PROGRAM MAIN
VAR
	master,slave:					axis_ref;(*定义两个虚轴*)
	camming_state:					camming_state;(*定义变量调用枚举体*)
	
	camin:							MC_CamIn;(*用于电子凸轮耦合功能块*)
	camout:							MC_CamOut;(*用于电子凸轮解耦功能块*)
	CamTableSelect_1:				MC_CamTableSelect;(*用于创建凸轮表*)
	cam_table1:						MC_CAM_REF;(*用于定义凸轮表*)
	table1:							ARRAY[1..5] OF MC_MotionFunctionPoint;(*用于定义电子凸轮表中的关键点，此例子中包含五个关键点*)
	CamInOut,CamOutOut,selectOut:	ST_McOutputs;(*用于绑定相关功能块输出接口*)
	
	move_velo_master:				MC_MoveVelocity;
	move_abs_slave:					MC_MoveAbsolute;
	MoveMasterOut:					ST_McOutputs;
	MoveSlaveOut:					ST_McOutputs;
	
	ResetSlave,ResetMaster:			MC_Reset;
	ResetMasterOut,ResetSlaveOut:	ST_McOutputs;
	master_actpos,slave_actpos: 	LREAL;
	
//   ADD  ReadMotionFunctionValues //
	ReadMotionFunctionValues:		MC_ReadMotionFunctionValues;
	bReadMotionFunctionValues: 		BOOL;
	readCamTable:					MC_CAM_REF;
	
	EndPosMaster: LREAL := 100;
	StartPosMaster: LREAL := 0;
	Increment: LREAL := 1;
	table_test: ARRAY[0..100, 0..1] OF LREAL;
	temp_M: UDINT;

END_VAR

(*用于更新轴状态*)
master();
slave();

power();
camming();
reset();
move_m_s();
table1_point();

Act_ReadMotionFunctionValues();

CASE camming_state OF
	
	state_init:(*程序初始化*)
	
		move_velo_master.Execute:=FALSE;
		ResetMaster.Execute:=FALSE;
		ResetSlave.Execute:=FALSE;
		camin.Execute:=FALSE;
		camout.Execute:=FALSE;
		camming_state:=state_power;
		
	state_power:(*主从轴使能*)
	
		IF master.NcToPlc.StateDWord.0 AND slave.NcToPlc.StateDWord.0 THEN
			camming_state:=state_forward;
		ELSIF master.Status.Error OR slave.Status.Error THEN
			camming_state:=state_error;
		END_IF
		
	state_forward:(*主轴100正转，从轴回0*)
	
		move_velo_master.Execute:=TRUE;
		move_abs_slave.Execute:=TRUE;
		IF master.Status.Moving AND move_abs_slave.Done THEN
			move_velo_master.Execute:=FALSE;
			move_abs_slave.Execute:=FALSE;
			camming_state:=state_pre_table1;
		END_IF
		IF master.Status.Error OR slave.Status.Error THEN 
			camming_state:=state_error;
		END_IF
	
	state_pre_table1:
	
		CamTableSelect_1.Execute:=TRUE;
		camin.CamTableID:=1;
		IF CamTableSelect_1.Done THEN
			camming_state:=state_camming1;
			CamTableSelect_1.Execute:=FALSE;
		END_IF
		IF master.Status.Error OR slave.Status.Error THEN
			camming_state:=state_error;
		END_IF
		
	state_camming1:(*主从轴耦合，实现电子凸轮表*)
	
		camin.Execute:=TRUE;
		IF camin.InSync THEN
			camin.Execute:=FALSE;
			camming_state:=camming_status;
		END_IF
		IF master.Status.Error OR slave.Status.Error THEN
			camming_state:=state_error;
		END_IF

	camming_status:(*耦合成功后，通过camming_status来读取主从轴位置*)	
		
		master_actpos:=master.NcToPlc.SetPos;
		slave_actpos:=slave.NcToPlc.SetPos;
		IF master.Status.Error OR slave.Status.Error THEN
			camming_state:=state_error;
		END_IF
		
	state_error:(*若出现轴报错,需要凸轮解耦，复位*)

		camout.Execute:=slave.Status.Coupled;(*先解耦*)
		IF NOT slave.Status.Coupled THEN
			IF master.Status.Error OR slave.Status.Error THEN
				camming_state:=state_reset;(*轴报错需要reset*)
			ELSE
				camming_state:=state_init;(*若功能块报错，不需要reset*)	
			END_IF
		END_IF
		
	state_reset:

		ResetMaster.Execute:=TRUE;
		CamTableSelect_1.Execute:=FALSE;
		ResetSlave.Execute:=TRUE;
		IF ResetMaster.Done AND ResetSlave.Done THEN
			camming_state:=state_init;
		ELSIF ResetMaster.Error OR ResetSlave.Error THEN
			camming_state:=state_init;	
		END_IF
				
END_CASE

ACTION ACT_ReadMotionFunctionValues:
ReadMotionFunctionValues(
	Execute:=bReadMotionFunctionValues , 
	CamTableID:=1 , 
	ValueSelectMask:= MC_VALUETYPE_POSITION , 
	StartPosMaster:= StartPosMaster, 
	EndPosMaster:= EndPosMaster, 
	Increment:= Increment, 
	Done=> , 
	Busy=> , 
	Error=> , 
	ErrorID=> , 
	CamTable:=readCamTable );
	
readCamTable.ArraySize:=SIZEOF(table_test);
readCamTable.NoOfColumns:=2;
temp_M:=LREAL_TO_UDINT((EndPosMaster- StartPosMaster)/ Increment);
readCamTable.NoOfRows:=100;
readCamTable.pArray:=ADR(table_test);
readCamTable.TableType:= MC_TABLETYPE_EQUIDISTANT;
END_ACTION

ACTION camming:
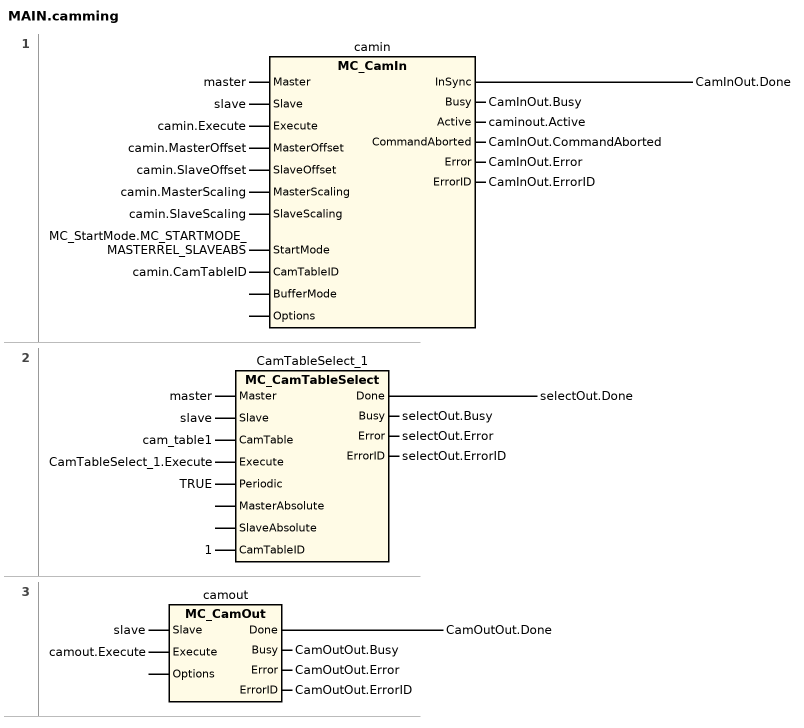
// NETWORK 1
camin(
    Master := master,
    Slave := slave,
    Execute := camin.Execute,
    MasterOffset := camin.MasterOffset,
    SlaveOffset := camin.SlaveOffset,
    MasterScaling := camin.MasterScaling,
    SlaveScaling := camin.SlaveScaling,
    StartMode := MC_StartMode.MC_STARTMODE_MASTERREL_SLAVEABS,
    CamTableID := camin.CamTableID,
    Busy => CamInOut.Busy,
    Active => caminout.Active,
    CommandAborted => CamInOut.CommandAborted,
    Error => CamInOut.Error,
    ErrorID => CamInOut.ErrorID); // MC_CamIn
CamInOut.Done := camin.InSync;

// NETWORK 2
CamTableSelect_1(
    Master := master,
    Slave := slave,
    CamTable := cam_table1,
    Execute := CamTableSelect_1.Execute,
    Periodic := TRUE,
    CamTableID := 1,
    Busy => selectOut.Busy,
    Error => selectOut.Error,
    ErrorID => selectOut.ErrorID); // MC_CamTableSelect
selectOut.Done := CamTableSelect_1.Done;

// NETWORK 3
camout(
    Slave := slave,
    Execute := camout.Execute,
    Busy => CamOutOut.Busy,
    Error => CamOutOut.Error,
    ErrorID => CamOutOut.ErrorID); // MC_CamOut
CamOutOut.Done := camout.Done;
END_ACTION

ACTION move_m_s:
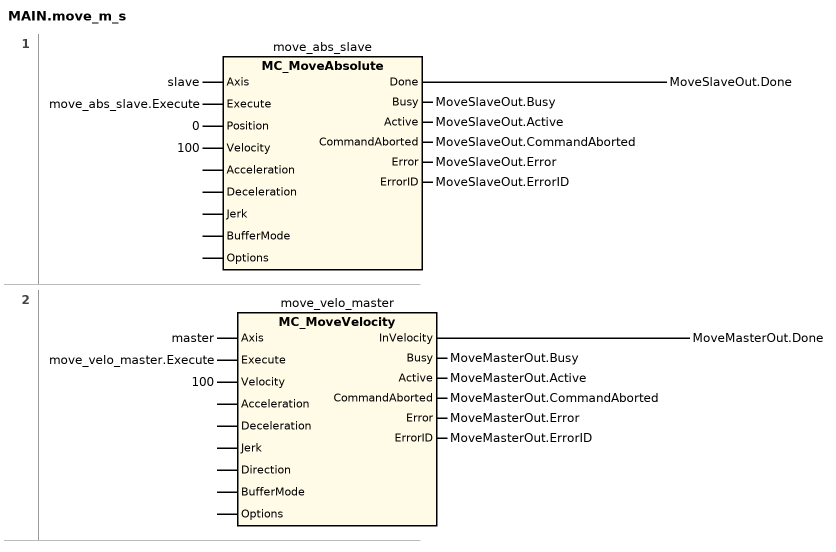
// NETWORK 1
move_abs_slave(
    Axis := slave,
    Execute := move_abs_slave.Execute,
    Position := 0,
    Velocity := 100,
    Busy => MoveSlaveOut.Busy,
    Active => MoveSlaveOut.Active,
    CommandAborted => MoveSlaveOut.CommandAborted,
    Error => MoveSlaveOut.Error,
    ErrorID => MoveSlaveOut.ErrorID); // MC_MoveAbsolute
MoveSlaveOut.Done := move_abs_slave.Done;

// NETWORK 2
move_velo_master(
    Axis := master,
    Execute := move_velo_master.Execute,
    Velocity := 100,
    Busy => MoveMasterOut.Busy,
    Active => MoveMasterOut.Active,
    CommandAborted => MoveMasterOut.CommandAborted,
    Error => MoveMasterOut.Error,
    ErrorID => MoveMasterOut.ErrorID); // MC_MoveVelocity
MoveMasterOut.Done := move_velo_master.InVelocity;
END_ACTION

ACTION power:
(*对两轴使能,同时设置速比*)

master.PlcToNc.ControlDWord:=7;
slave.PlcToNc.ControlDWord:=7;

master.PlcToNc.Override:=1000000;
slave.PlcToNc.Override:=1000000;
END_ACTION

ACTION reset:
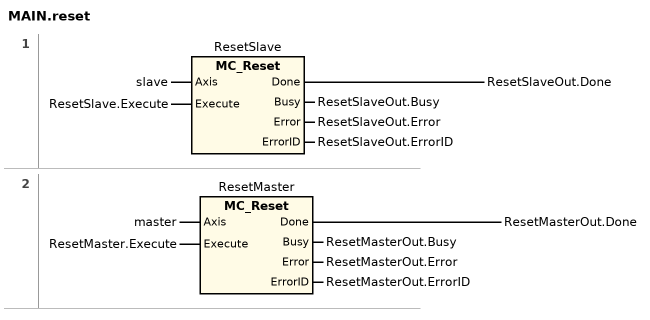
// NETWORK 1
ResetSlave(
    Axis := slave,
    Execute := ResetSlave.Execute,
    Busy => ResetSlaveOut.Busy,
    Error => ResetSlaveOut.Error,
    ErrorID => ResetSlaveOut.ErrorID); // MC_Reset
ResetSlaveOut.Done := ResetSlave.Done;

// NETWORK 2
ResetMaster(
    Axis := master,
    Execute := ResetMaster.Execute,
    Busy => ResetMasterOut.Busy,
    Error => ResetMasterOut.Error,
    ErrorID => ResetMasterOut.ErrorID); // MC_Reset
ResetMasterOut.Done := ResetMaster.Done;
END_ACTION

ACTION table1_point:
cam_table1.ArraySize:=SIZEOF(table1);
cam_table1.NoOfColumns:=1;
cam_table1.NoOfRows:=5;
cam_table1.pArray:=ADR(table1);
cam_table1.TableType:=MC_TABLETYPE_MOTIONFUNCTION;


table1[1].FunctionType:=MOTIONFUNCTYPE_POLYNOM5;
table1[1].MasterPos:=0;
table1[1].SlavePos:=0;
table1[1].PointIndex:=1;
table1[1].PointType:=MOTIONPOINTTYPE_MOTION;

table1[2].FunctionType:=MOTIONFUNCTYPE_POLYNOM5;
table1[2].MasterPos:=90;
table1[2].SlavePos:=100;
table1[2].PointIndex:=2;
table1[2].PointType:=MOTIONPOINTTYPE_MOTION;

table1[3].FunctionType:=MOTIONFUNCTYPE_POLYNOM5;
table1[3].MasterPos:=180;
table1[3].SlavePos:=80;
table1[3].PointIndex:=3;
table1[3].PointType:=MOTIONPOINTTYPE_MOTION;

table1[4].FunctionType:=MOTIONFUNCTYPE_POLYNOM5;
table1[4].MasterPos:=270;
table1[4].SlavePos:=50;
table1[4].PointIndex:=4;
table1[4].PointType:=MOTIONPOINTTYPE_MOTION;

table1[5].FunctionType:=MOTIONFUNCTYPE_POLYNOM5;
table1[5].MasterPos:=360;
table1[5].SlavePos:=0;
table1[5].PointIndex:=5;
table1[5].PointType:=MOTIONPOINTTYPE_MOTION;
END_ACTION

END_PROGRAM

(* stored: Version 1.1.0.1, ProductVersion 3.1.4024.10
   POU MAIN: Id {97635362-d819-4a9a-8783-11f895aa8470}, SpecialFunc None
   Action ACT_ReadMotionFunctionValues: Id {57e81dff-27ee-4eeb-8238-62ec7519236b}
   Action camming: Id {2bbcdff9-b2da-4030-84d5-557527ce74cc}
   Action move_m_s: Id {9d3da378-3c7c-4dbd-bbf0-b652e2972c78}
   Action power: Id {1a264cdc-f98a-4dc2-b2f4-d4d8cc3cd6e9}
   Action reset: Id {1179c873-b2ec-468f-8124-9c26fdc0f0c1}
   Action table1_point: Id {b82b114b-242e-4378-9a33-62f360bdba26} *)
